(* Logix 5000 project; controller code_tcc vendor 1 type 14 code 106 rev 33.11; software revision 33.01 *)

TASK MainTask (periodic, rate 10 ms, priority 1, watchdog 500 ms) : MainProgram

MODULES
   Local : vendor 1 type 14 code 106 (Compact 0, rev 33.11)
END_MODULES

TYPE raC_UDT_ModbusClientConnection :
STRUCT
   LocalSlot : SINT;   // Local Slot for Ethernet module. For ControlLogix - L8x, EN2T(R) - use the actual module slot. For CompactLogix use slot 0.
   LocalAddress : STR0016;   // Used only for controllers with more than 1 local IP address (5380, 5480). For all others must be blank.
   DestAddress : STR0016;   // The IP address for the Modbus TCP Slave device to connect to
   DestinationPort : DINT;   // Default Modbus is 502
   MSG_Src : SINT[500];   // Placeholder for message source
   MSG_Dest : SINT[500];   // Placeholder for message destination
END_STRUCT
END_TYPE

TYPE raC_UDT_ModbusClientData :
STRUCT
   Coils_0xxx : BOOL[1024];
   DiscInputs_1xxx : BOOL[1024];
   InpRegisters_3xxx : INT[1024];
   HoldRegisters_4xxx : INT[1024];
END_STRUCT
END_TYPE

TYPE raC_UDT_ModbusClientHMI :
STRUCT
   Parameters : raC_UDT_ModbusClientConnection;
   Transaction : raC_UDT_ModbusClientTransaction;
   Index0x : DINT;
   Index1x : DINT;
   Index3x : DINT;
   Index4x : DINT;
   DataValue : INT[65];
   DataAddr : DINT[65];
   TransactionIndex : DINT;
   RemoteAddrStart : DINT;
   RemoteAddrEnd : DINT;
   LocalAddrEnd : DINT;
END_STRUCT
END_TYPE

TYPE raC_UDT_ModbusClientTransaction :
STRUCT
   Enabled : BOOL;   // Enables (1) or disables (0) the transaction
   PollInterval : DINT;   // Time between triggers in milliseconds. Minimum is 80 msec. Anyting below 80 will be set to 1 seconds
   TransType : INT;   // Transaction code for the Modbus Protocol. Acceptable values are 1-Coil Read, 2- Discrete Input read, 3-Holding Register Read, 4-Input Register Read, 5-Write Single Coil, 6-Single Holding Register Write, 15-Multiple Coil Write, 16 Multiple Holding Register Write
   StationID : SINT;   // Station ID ( Unit Identifier). Commonly used if going through a gateway or bridge in which case it is the device address on the other side of the gateway. Other wise leave as 0
   BeginAddress : DINT;   // Beginning address in remote device to read from or write to.
   Count : INT;   // The number of items in remote device to read from or write to.
   LocalAddress : INT;   // Beginning address in in this programs' "_Data" arrays
   TransComplete : BOOL;   // Transaction Complete Flag. Check the TransStat to see if the transaction was successful or if a Modbus exception code was returned.
   TransStat : INT;   // Status result of the transaction. 0 = success, 1 = in process 2 = retry -1 = exception
   Diagnostic : raC_UDT_ModbusClientTransactionDiag;
END_STRUCT
END_TYPE

TYPE raC_UDT_ModbusClientTransactionDiag :
STRUCT
   Request : STR0500;   // Actual buffer used to build the modbus request that is transmited to the remote node.
   ReqBuilt : BOOL;   // Transaction request string is built, clear this if anything is changed in a read operation to rebuild the Request string.
   Overlap : BOOL;   // Transaction is not completing before next trigger
   Overload : BOOL;   // Transaction is not completing because of excessive Overlaps in one or more transactions
   TransID : INT;   // Serial Number of the actual Ethernet Transaction used to match to the appropriate Reply
   TransLastError : INT;   // Last Error on transaction. 0-Success, -2 Network write error, -3 Local write error, -4 Network Read Error, -5 Local Read Error, -6 Connection failed.. -12 Invalid Trans code, -13 Out of data array range.
   IntervalTimer : TIMER;   // IntervalTimer, used to trigger transaction
   NoReplyCounter : COUNTER;   // No Reply Counter
   PendingTimer : TIMER;   // Timing pending requests
END_STRUCT
END_TYPE

TYPE raC_UDT_ModbusConnectParam :   // Parameterss for the OpenConnection Service
STRUCT
   Timeout : DINT;
   DestAddr : STR0032;
END_STRUCT
END_TYPE

TYPE raC_UDT_ModbusCreateParam :
STRUCT
   Type : DINT;   // Type 1-TCP, 2-UDP
   Family : INT;   // Address Family Must be 2
   Port : INT;   // Local Port Number
   Addr : DINT;   // Local IP Address
END_STRUCT
END_TYPE

TYPE STR0008 :
STRUCT
   LEN : DINT;
   DATA : SINT[8];
END_STRUCT
END_TYPE

TYPE STR0016 :
STRUCT
   LEN : DINT;
   DATA : SINT[16];
END_STRUCT
END_TYPE

TYPE STR0032 :
STRUCT
   LEN : DINT;
   DATA : SINT[32];
END_STRUCT
END_TYPE

TYPE STR0500 :
STRUCT
   LEN : DINT;
   DATA : SINT[500];
END_STRUCT
END_TYPE

TYPE STR4096 :
STRUCT
   LEN : DINT;
   DATA : SINT[4096];
END_STRUCT
END_TYPE

ADD_ON_INSTRUCTION raC_Opr_NetModbusTCPClient   (* revision 2.4 0, ExecutePrescan *)
// Modbus TCP Client
// Revision note:
// 2.0.0 Initial Release in AOI format
// 2.0.1 Corrected local IP address logic
// 2.1.0 Corrected Overload and Overlap indicators
// 2.2.0 Changed BeginAddress from INT to DINT, force LocalSlot 0 for CompactLogix
// 2.3.0 HMI interface
// 2.4.0 Improved malformed packet handling
VAR_INPUT
   Inp_Enable : BOOL; {required}
END_VAR
VAR_IN_OUT
   Ref_Connection : raC_UDT_ModbusClientConnection; {required}
   Ref_Transactions : raC_UDT_ModbusClientTransaction[5]; {required}
   Ref_ModbusData : raC_UDT_ModbusClientData; {required}
   Ref_MsgCreate : MESSAGE; {required}
   Ref_MsgConnect : MESSAGE; {required}
   Ref_MsgRead : MESSAGE; {required}
   Ref_MsgWrite : MESSAGE; {required}
   Ref_MsgDelete : MESSAGE; {required}
   Ref_MsgSetAttrSingle : MESSAGE; {required}
END_VAR
VAR_OUTPUT
   Sts_EN : BOOL; {access Read Only, visible}
   Sts_Connected : BOOL; {access Read Only, visible}
   Sts_Faulted : BOOL; {access Read Only, visible}
   Sts_Overlap : BOOL; {access Read Only, visible}
   Sts_Overload : BOOL; {access Read Only, visible}
   Sts_LastError : DINT; {access Read Only}   // The last recorded socket error for this connection. 0 good, -2 Write Error, -4 Read Error, -6 connection failed, -7 Delete all failed, -8 Create Soc failed, -9 Connection failed, -10 connection dropped, -11 error in setting socket parameter. -12 - Enable removed
END_VAR
VAR
   Wrk_MSGStep : DINT; {access None}
   Wrk_CreateReq : raC_UDT_ModbusCreateParam; {access None}
   Wrk_Instance : DINT; {access None}
   Wrk_ConnectReq : raC_UDT_ModbusConnectParam; {access None}
   Wrk_PortStr : STR0016 := '?port='; {access None}
   Wrk_TempStr : STR0016; {access None}
   Wrk_RetryTimer : TIMER := (PRE := 5000); {access None}
   Wrk_MSGRead_SRC : DINT[2]; {access None}   // User for MSG Read Source
   Wrk_TempString : STR0500; {access None}
   Wrk_Main_Read_Buffer : STR4096; {access None}
   Wrk_WrIndex : DINT; {access None}
   Wrk_TransactionTriggers : BOOL[32]; {access None}
   Wrk_BRS : raC_Tec_NetModbusTCPClient_BuildReqStr; {access None}
   Wrk_IDCounter : DINT; {access None}
   Wrk_WriteNow : BOOL[32]; {access None}   // Transmit Request Flags
   Wrk_TempDINT : DINT; {access None}
   Wrk_AdditionalLen : INT; {access None}
   Wrk_ModbusTransID : INT; {access None}
   Wrk_AdditionaLenRead : INT; {access None}
   Wrk_ModbusCmdLen : INT; {access None}
   Wrk_ModbusPacket : STR0500; {access None}
   Wrk_DataReceived : BOOL; {access None}
   Wrk_CmdFromReadPacket : DINT; {access None}
   Wrk_ModbusID : STR0008; {access None}
   Wrk_AdditionalLen1 : INT; {access None}
   Wrk_ModbusCmdTemp : INT; {access None}
   Wrk_ModbusUnit : STR0008; {access None}
   Wrk_ModbusBytes : DINT; {access None}
   Wrk_ModbusCmdString : STR0500; {access None}
   Wrk_CWR : raC_Tec_NetModbusTCPClient_ChkWrReply; {access None}
   Wrk_RSB : raC_Tec_NetModbusTCPClient_RespStrBit; {access None}
   Wrk_TransIndex : DINT; {access None}
   Wrk_TimerIndex : DINT; {access None}
   Wrk_ArraySize : DINT; {access None}
   Wrk_LastTransaction : DINT; {access None}
   Wrk_RSW : raC_Tec_NetModbusTCPClient_RespStrWord; {access None}
   Wrk_TempOctet : DINT[4]; {access None}
   Wrk_TempStrOctet : STR0008; {access None}
   Wrk_TempStrOctetlen : DINT; {access None}
   Wrk_TempIPStr : STR0016; {access None}
   Wrk_TempInt : DINT; {access None}
   Wrk_ClrReqIndex : DINT; {access None}
   Wrk_StepLockTimer : TIMER := (PRE := 10000); {access None}
   Wrk_Controller_Name : SINT[33]; {access None}
   Wrk_Controller_Type : DINT; {access None}
   Wrk_InitCompleted : BOOL; {access None}
   Inf_Lib : STR0016; {access Read Only}
   Inf_Type : STR0032; {access Read Only}
   Inf_Version : STR0016; {access Read Only}
   HMI_Tab : DINT;
   Wrk_tempHMItransaction : DINT; {access None}
   Wrk_HMITransactionValid : BOOL; {access None}
   wrk_FAL_Addr : CONTROL := (LEN := 64); {access None}
   wrk_LoopIndex : DINT; {access None}
   wrk_AddrIndex : DINT; {access None}
   HMI : raC_UDT_ModbusClientHMI;
   Wrk_OLindex : DINT; {access None}
   Wrk_OverloadStatus : BOOL; {access None}
   Wrk_OverlapStatus : BOOL; {access None}
END_VAR

ROUTINE Logic   (* ladder *)
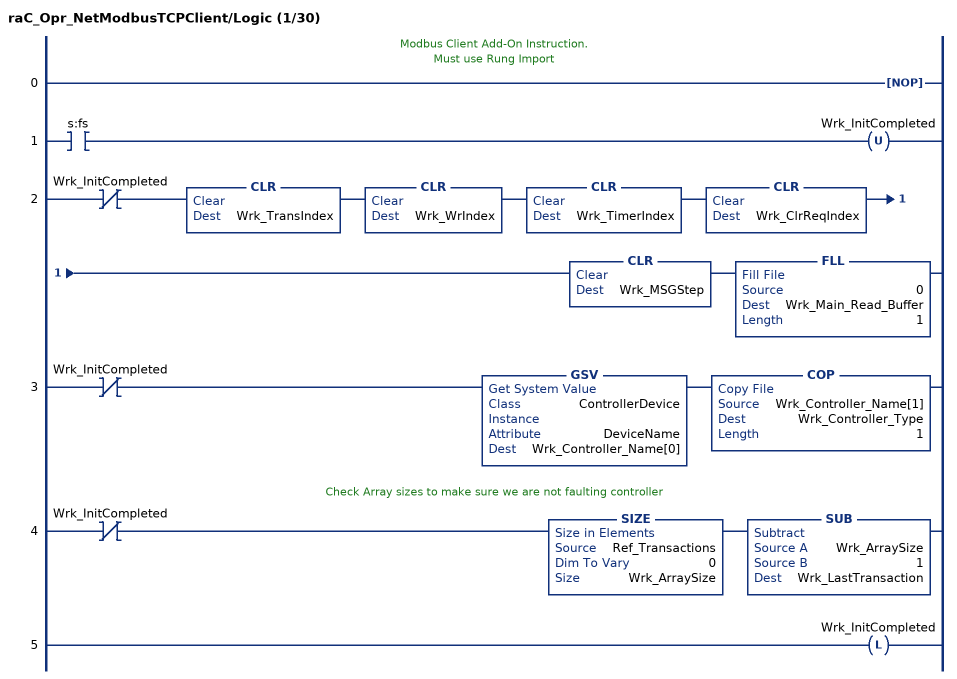
   // Modbus Client Add-On Instruction.
   // Must use Rung Import
   0: NOP();
   1: XIC(s:fs)OTU(Wrk_InitCompleted);
   2: XIO(Wrk_InitCompleted)CLR(Wrk_TransIndex)CLR(Wrk_WrIndex)CLR(Wrk_TimerIndex)CLR(Wrk_ClrReqIndex)CLR(Wrk_MSGStep)FLL(0,Wrk_Main_Read_Buffer,1);
   3: XIO(Wrk_InitCompleted)GSV(ControllerDevice,,DeviceName,Wrk_Controller_Name[0])COP(Wrk_Controller_Name[1],Wrk_Controller_Type,1);
   // Check Array sizes to make sure we are not faulting controller
   4: XIO(Wrk_InitCompleted)SIZE(Ref_Transactions,0,Wrk_ArraySize)SUB(Wrk_ArraySize,1,Wrk_LastTransaction);
   5: OTL(Wrk_InitCompleted);
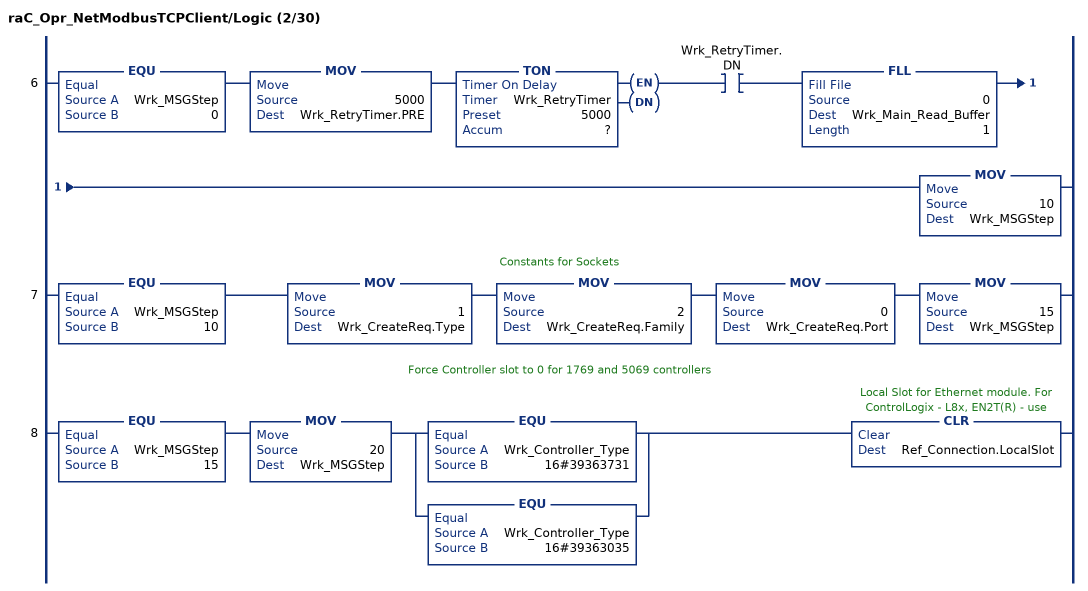
   6: EQU(Wrk_MSGStep,0)MOV(5000,Wrk_RetryTimer.PRE)TON(Wrk_RetryTimer,?,?)XIC(Wrk_RetryTimer.DN)FLL(0,Wrk_Main_Read_Buffer,1)MOV(10,Wrk_MSGStep);
   // Constants for Sockets
   7: EQU(Wrk_MSGStep,10)MOV(1,Wrk_CreateReq.Type)MOV(2,Wrk_CreateReq.Family)MOV(0,Wrk_CreateReq.Port)MOV(15,Wrk_MSGStep);
   // Force Controller slot to 0 for 1769 and 5069 controllers
   8: EQU(Wrk_MSGStep,15)MOV(20,Wrk_MSGStep)[EQU(Wrk_Controller_Type,16#39363731) ,EQU(Wrk_Controller_Type,16#39363035) ]CLR(Ref_Connection.LocalSlot);
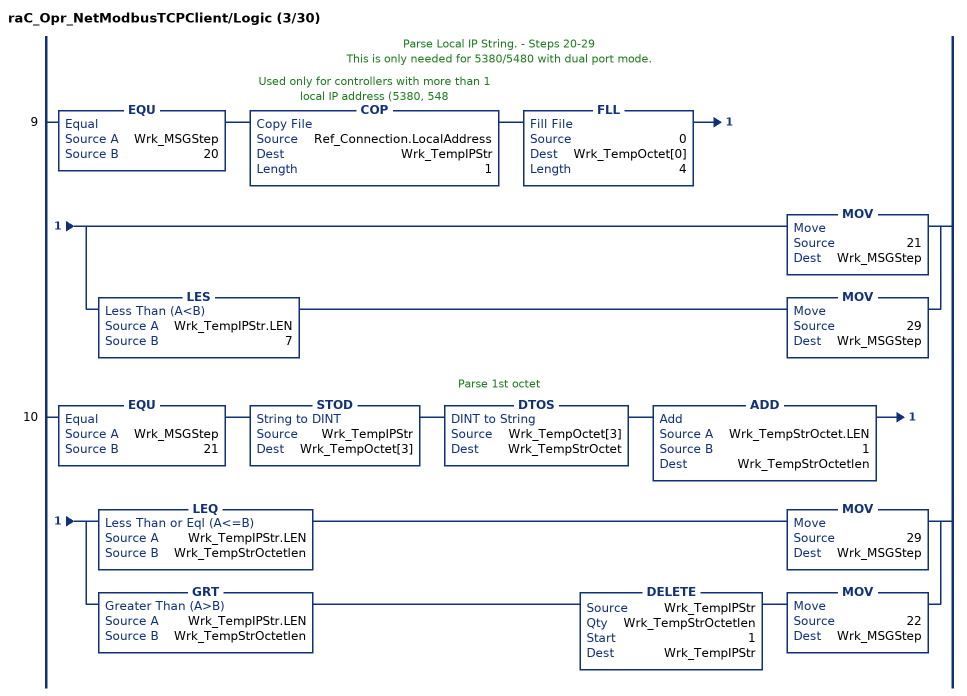
   // Parse Local IP String. - Steps 20-29
   // This is only needed for 5380/5480 with dual port mode.
   9: EQU(Wrk_MSGStep,20)COP(Ref_Connection.LocalAddress,Wrk_TempIPStr,1)FLL(0,Wrk_TempOctet[0],4)[MOV(21,Wrk_MSGStep) ,LES(Wrk_TempIPStr.LEN,7) MOV(29,Wrk_MSGStep) ];
   // Parse 1st octet
   10: EQU(Wrk_MSGStep,21)STOD(Wrk_TempIPStr,Wrk_TempOctet[3])DTOS(Wrk_TempOctet[3],Wrk_TempStrOctet)ADD(Wrk_TempStrOctet.LEN,1,Wrk_TempStrOctetlen)[LEQ(Wrk_TempIPStr.LEN,Wrk_TempStrOctetlen) MOV(29,Wrk_MSGStep) ,GRT(Wrk_TempIPStr.LEN,Wrk_TempStrOctetlen) DELETE(Wrk_TempIPStr,Wrk_TempStrOctetlen,1,Wrk_TempIPStr) MOV(22,Wrk_MSGStep) ];
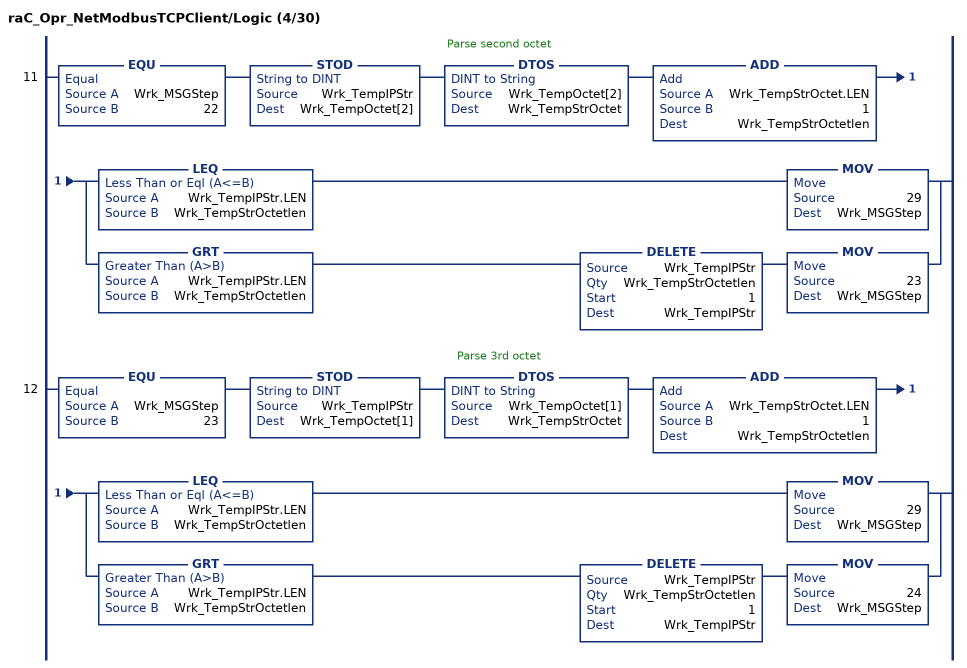
   // Parse second octet
   11: EQU(Wrk_MSGStep,22)STOD(Wrk_TempIPStr,Wrk_TempOctet[2])DTOS(Wrk_TempOctet[2],Wrk_TempStrOctet)ADD(Wrk_TempStrOctet.LEN,1,Wrk_TempStrOctetlen)[LEQ(Wrk_TempIPStr.LEN,Wrk_TempStrOctetlen) MOV(29,Wrk_MSGStep) ,GRT(Wrk_TempIPStr.LEN,Wrk_TempStrOctetlen) DELETE(Wrk_TempIPStr,Wrk_TempStrOctetlen,1,Wrk_TempIPStr) MOV(23,Wrk_MSGStep) ];
   // Parse 3rd octet
   12: EQU(Wrk_MSGStep,23)STOD(Wrk_TempIPStr,Wrk_TempOctet[1])DTOS(Wrk_TempOctet[1],Wrk_TempStrOctet)ADD(Wrk_TempStrOctet.LEN,1,Wrk_TempStrOctetlen)[LEQ(Wrk_TempIPStr.LEN,Wrk_TempStrOctetlen) MOV(29,Wrk_MSGStep) ,GRT(Wrk_TempIPStr.LEN,Wrk_TempStrOctetlen) DELETE(Wrk_TempIPStr,Wrk_TempStrOctetlen,1,Wrk_TempIPStr) MOV(24,Wrk_MSGStep) ];
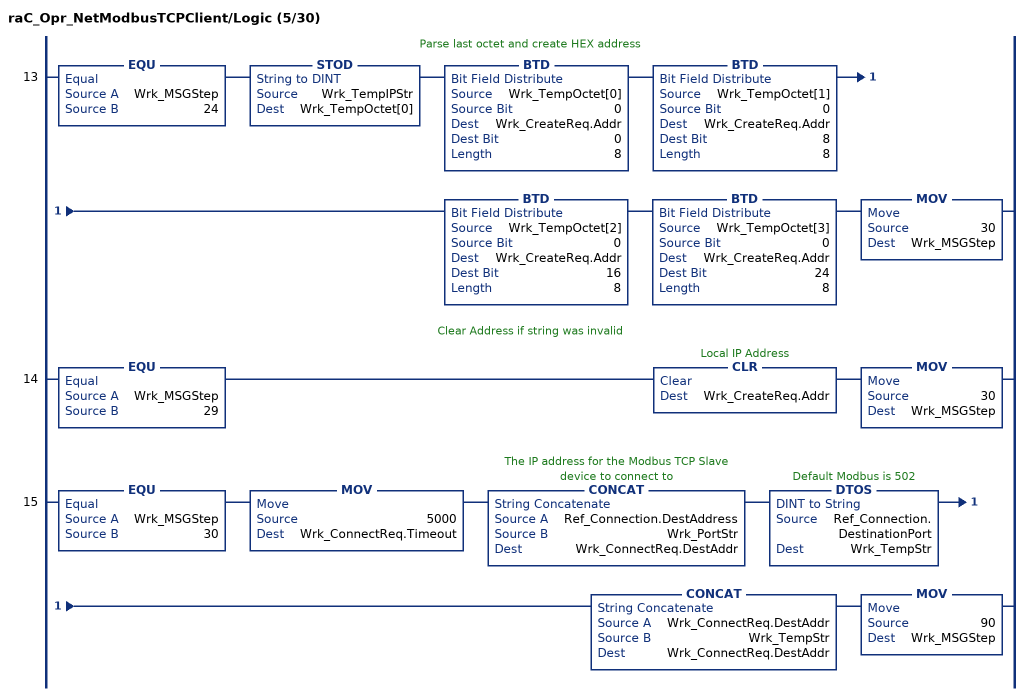
   // Parse last octet and create HEX address
   13: EQU(Wrk_MSGStep,24)STOD(Wrk_TempIPStr,Wrk_TempOctet[0])BTD(Wrk_TempOctet[0],0,Wrk_CreateReq.Addr,0,8)BTD(Wrk_TempOctet[1],0,Wrk_CreateReq.Addr,8,8)BTD(Wrk_TempOctet[2],0,Wrk_CreateReq.Addr,16,8)BTD(Wrk_TempOctet[3],0,Wrk_CreateReq.Addr,24,8)MOV(30,Wrk_MSGStep);
   // Clear Address if string was invalid
   14: EQU(Wrk_MSGStep,29)CLR(Wrk_CreateReq.Addr)MOV(30,Wrk_MSGStep);
   15: EQU(Wrk_MSGStep,30)MOV(5000,Wrk_ConnectReq.Timeout)CONCAT(Ref_Connection.DestAddress,Wrk_PortStr,Wrk_ConnectReq.DestAddr)DTOS(Ref_Connection.DestinationPort,Wrk_TempStr)CONCAT(Wrk_ConnectReq.DestAddr,Wrk_TempStr,Wrk_ConnectReq.DestAddr)MOV(90,Wrk_MSGStep);
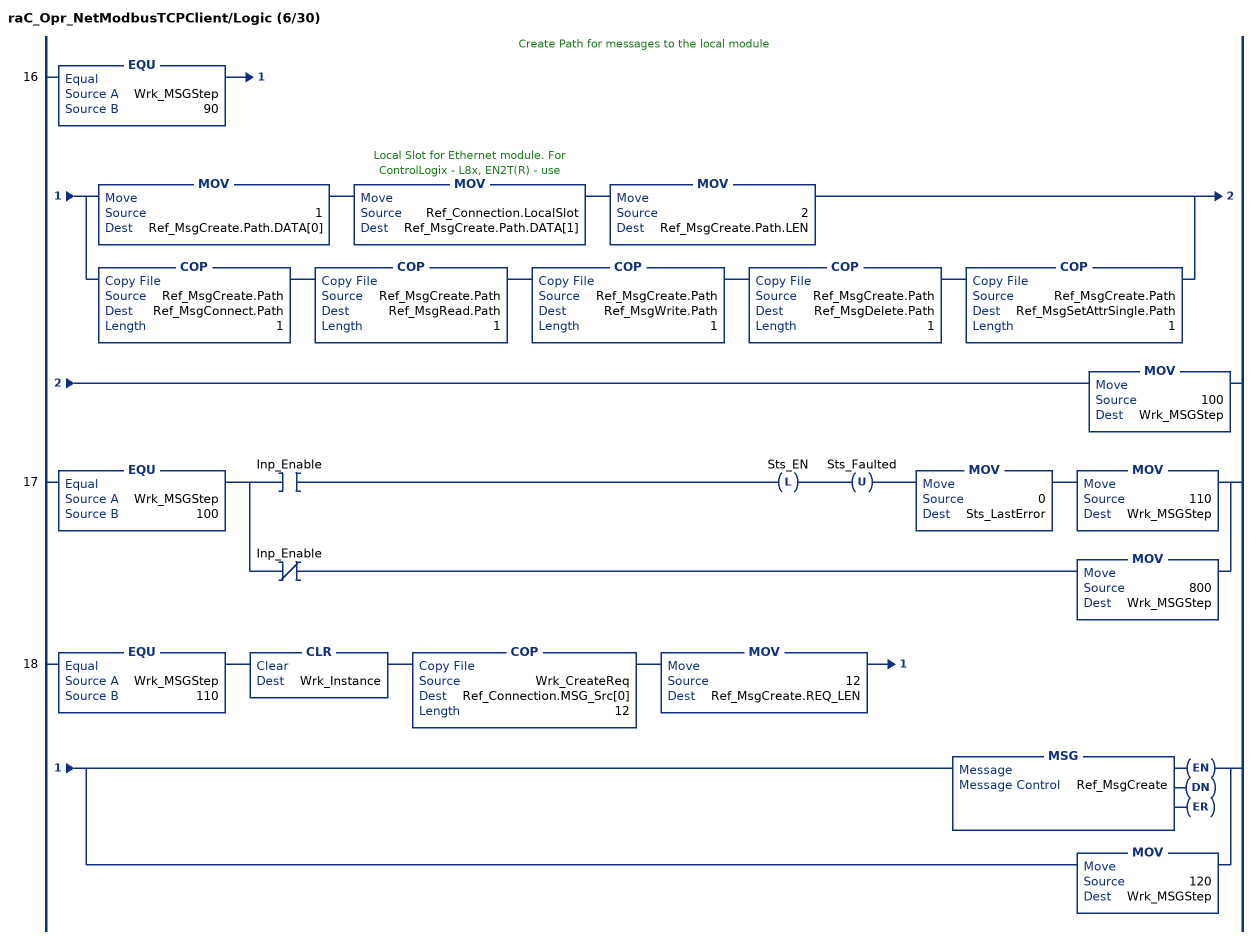
   // Create Path for messages to the local module
   16: EQU(Wrk_MSGStep,90)[MOV(1,Ref_MsgCreate.Path.DATA[0]) MOV(Ref_Connection.LocalSlot,Ref_MsgCreate.Path.DATA[1]) MOV(2,Ref_MsgCreate.Path.LEN) ,COP(Ref_MsgCreate.Path,Ref_MsgConnect.Path,1) COP(Ref_MsgCreate.Path,Ref_MsgRead.Path,1) COP(Ref_MsgCreate.Path,Ref_MsgWrite.Path,1) COP(Ref_MsgCreate.Path,Ref_MsgDelete.Path,1) COP(Ref_MsgCreate.Path,Ref_MsgSetAttrSingle.Path,1) ]MOV(100,Wrk_MSGStep);
   17: EQU(Wrk_MSGStep,100)[XIC(Inp_Enable) OTL(Sts_EN) OTU(Sts_Faulted) MOV(0,Sts_LastError) MOV(110,Wrk_MSGStep) ,XIO(Inp_Enable) MOV(800,Wrk_MSGStep) ];
   18: EQU(Wrk_MSGStep,110)CLR(Wrk_Instance)COP(Wrk_CreateReq,Ref_Connection.MSG_Src[0],12)MOV(12,Ref_MsgCreate.REQ_LEN)[MSG(Ref_MsgCreate) ,MOV(120,Wrk_MSGStep) ];
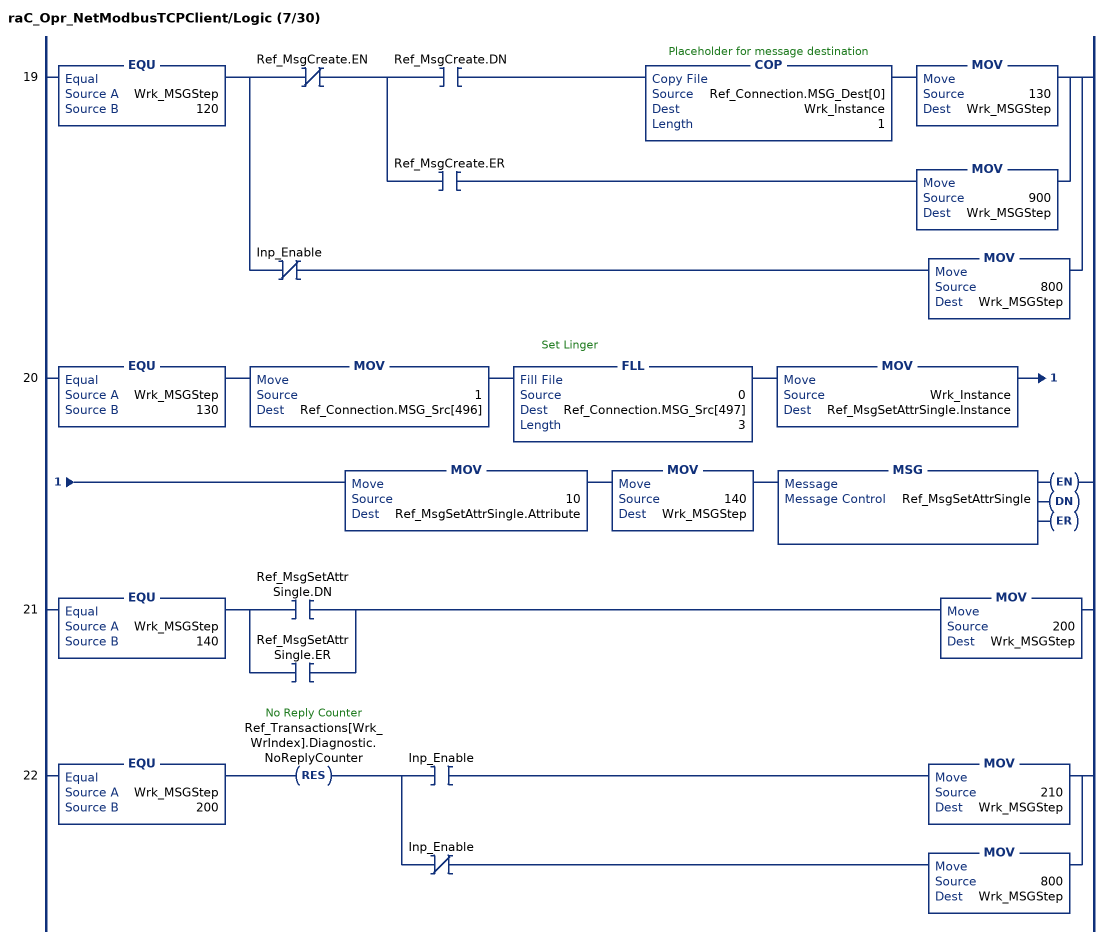
   19: EQU(Wrk_MSGStep,120)[XIO(Ref_MsgCreate.EN) [XIC(Ref_MsgCreate.DN) COP(Ref_Connection.MSG_Dest[0],Wrk_Instance,1) MOV(130,Wrk_MSGStep) ,XIC(Ref_MsgCreate.ER) MOV(900,Wrk_MSGStep) ] ,XIO(Inp_Enable) MOV(800,Wrk_MSGStep) ];
   // Set Linger
   20: EQU(Wrk_MSGStep,130)MOV(1,Ref_Connection.MSG_Src[496])FLL(0,Ref_Connection.MSG_Src[497],3)MOV(Wrk_Instance,Ref_MsgSetAttrSingle.Instance)MOV(10,Ref_MsgSetAttrSingle.Attribute)MOV(140,Wrk_MSGStep)MSG(Ref_MsgSetAttrSingle);
   21: EQU(Wrk_MSGStep,140)[XIC(Ref_MsgSetAttrSingle.DN) ,XIC(Ref_MsgSetAttrSingle.ER) ]MOV(200,Wrk_MSGStep);
   22: EQU(Wrk_MSGStep,200)RES(Ref_Transactions[Wrk_WrIndex].Diagnostic.NoReplyCounter)[XIC(Inp_Enable) MOV(210,Wrk_MSGStep) ,XIO(Inp_Enable) MOV(800,Wrk_MSGStep) ];
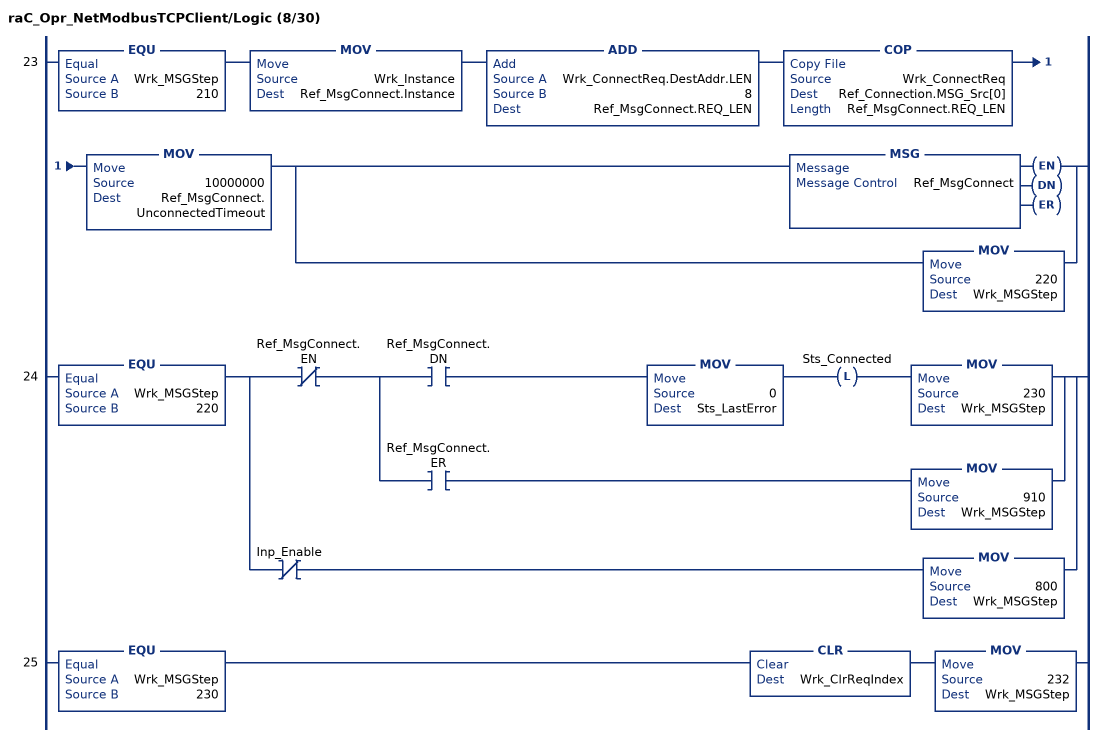
   23: EQU(Wrk_MSGStep,210)MOV(Wrk_Instance,Ref_MsgConnect.Instance)ADD(Wrk_ConnectReq.DestAddr.LEN,8,Ref_MsgConnect.REQ_LEN)COP(Wrk_ConnectReq,Ref_Connection.MSG_Src[0],Ref_MsgConnect.REQ_LEN)MOV(10000000,Ref_MsgConnect.UnconnectedTimeout)[MSG(Ref_MsgConnect) ,MOV(220,Wrk_MSGStep) ];
   24: EQU(Wrk_MSGStep,220)[XIO(Ref_MsgConnect.EN) [XIC(Ref_MsgConnect.DN) MOV(0,Sts_LastError) OTL(Sts_Connected) MOV(230,Wrk_MSGStep) ,XIC(Ref_MsgConnect.ER) MOV(910,Wrk_MSGStep) ] ,XIO(Inp_Enable) MOV(800,Wrk_MSGStep) ];
   25: EQU(Wrk_MSGStep,230)CLR(Wrk_ClrReqIndex)MOV(232,Wrk_MSGStep);
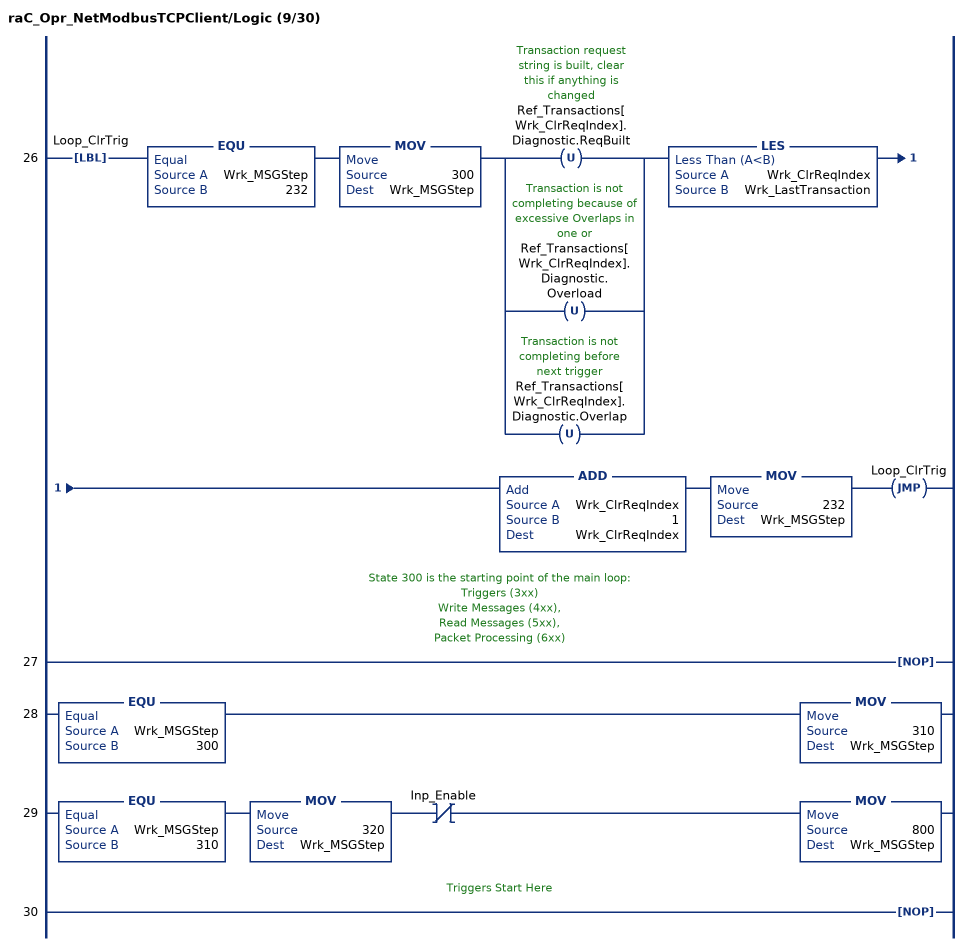
   26: LBL(Loop_ClrTrig)EQU(Wrk_MSGStep,232)MOV(300,Wrk_MSGStep)[OTU(Ref_Transactions[Wrk_ClrReqIndex].Diagnostic.ReqBuilt) ,OTU(Ref_Transactions[Wrk_ClrReqIndex].Diagnostic.Overload) ,OTU(Ref_Transactions[Wrk_ClrReqIndex].Diagnostic.Overlap) ]LES(Wrk_ClrReqIndex,Wrk_LastTransaction)ADD(Wrk_ClrReqIndex,1,Wrk_ClrReqIndex)MOV(232,Wrk_MSGStep)JMP(Loop_ClrTrig);
   // State 300 is the starting point of the main loop:
   // Triggers (3xx)
   // Write Messages (4xx),
   // Read Messages (5xx),
   // Packet Processing (6xx)
   27: NOP();
   28: EQU(Wrk_MSGStep,300)MOV(310,Wrk_MSGStep);
   29: EQU(Wrk_MSGStep,310)MOV(320,Wrk_MSGStep)XIO(Inp_Enable)MOV(800,Wrk_MSGStep);
   // Triggers Start Here
   30: NOP();
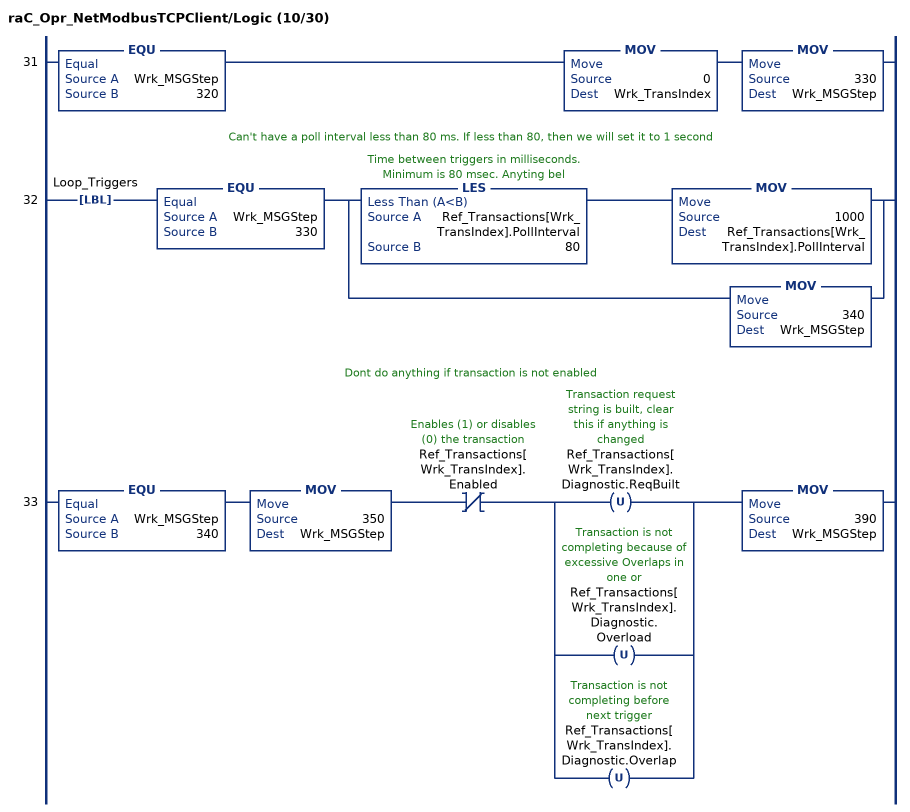
   31: EQU(Wrk_MSGStep,320)MOV(0,Wrk_TransIndex)MOV(330,Wrk_MSGStep);
   // Can't have a poll interval less than 80 ms. If less than 80, then we will set it to 1 second
   32: LBL(Loop_Triggers)EQU(Wrk_MSGStep,330)[LES(Ref_Transactions[Wrk_TransIndex].PollInterval,80) MOV(1000,Ref_Transactions[Wrk_TransIndex].PollInterval) ,MOV(340,Wrk_MSGStep) ];
   // Dont do anything if transaction is not enabled
   33: EQU(Wrk_MSGStep,340)MOV(350,Wrk_MSGStep)XIO(Ref_Transactions[Wrk_TransIndex].Enabled)[OTU(Ref_Transactions[Wrk_TransIndex].Diagnostic.ReqBuilt) ,OTU(Ref_Transactions[Wrk_TransIndex].Diagnostic.Overload) ,OTU(Ref_Transactions[Wrk_TransIndex].Diagnostic.Overlap) ]MOV(390,Wrk_MSGStep);
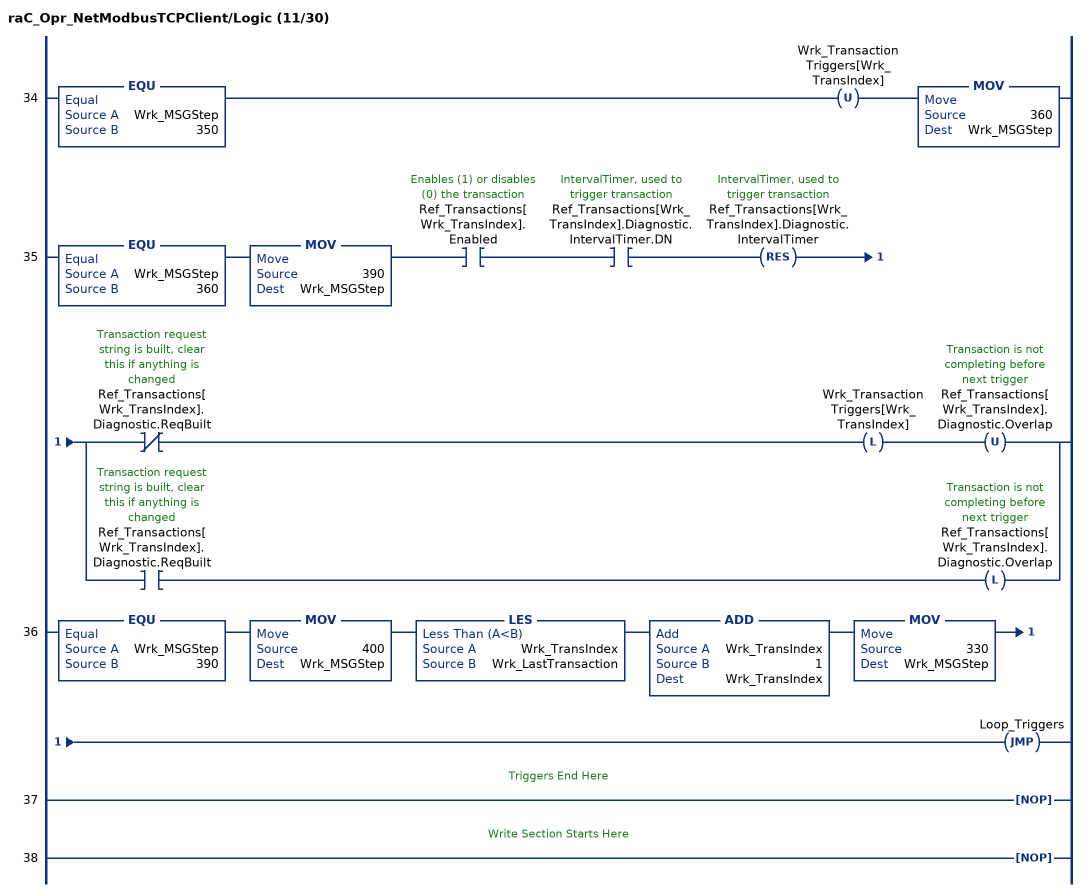
   34: EQU(Wrk_MSGStep,350)OTU(Wrk_TransactionTriggers[Wrk_TransIndex])MOV(360,Wrk_MSGStep);
   35: EQU(Wrk_MSGStep,360)MOV(390,Wrk_MSGStep)XIC(Ref_Transactions[Wrk_TransIndex].Enabled)XIC(Ref_Transactions[Wrk_TransIndex].Diagnostic.IntervalTimer.DN)RES(Ref_Transactions[Wrk_TransIndex].Diagnostic.IntervalTimer)[XIO(Ref_Transactions[Wrk_TransIndex].Diagnostic.ReqBuilt) OTL(Wrk_TransactionTriggers[Wrk_TransIndex]) OTU(Ref_Transactions[Wrk_TransIndex].Diagnostic.Overlap) ,XIC(Ref_Transactions[Wrk_TransIndex].Diagnostic.ReqBuilt) OTL(Ref_Transactions[Wrk_TransIndex].Diagnostic.Overlap) ];
   36: EQU(Wrk_MSGStep,390)MOV(400,Wrk_MSGStep)LES(Wrk_TransIndex,Wrk_LastTransaction)ADD(Wrk_TransIndex,1,Wrk_TransIndex)MOV(330,Wrk_MSGStep)JMP(Loop_Triggers);
   // Triggers End Here
   37: NOP();
   // Write Section Starts Here
   38: NOP();
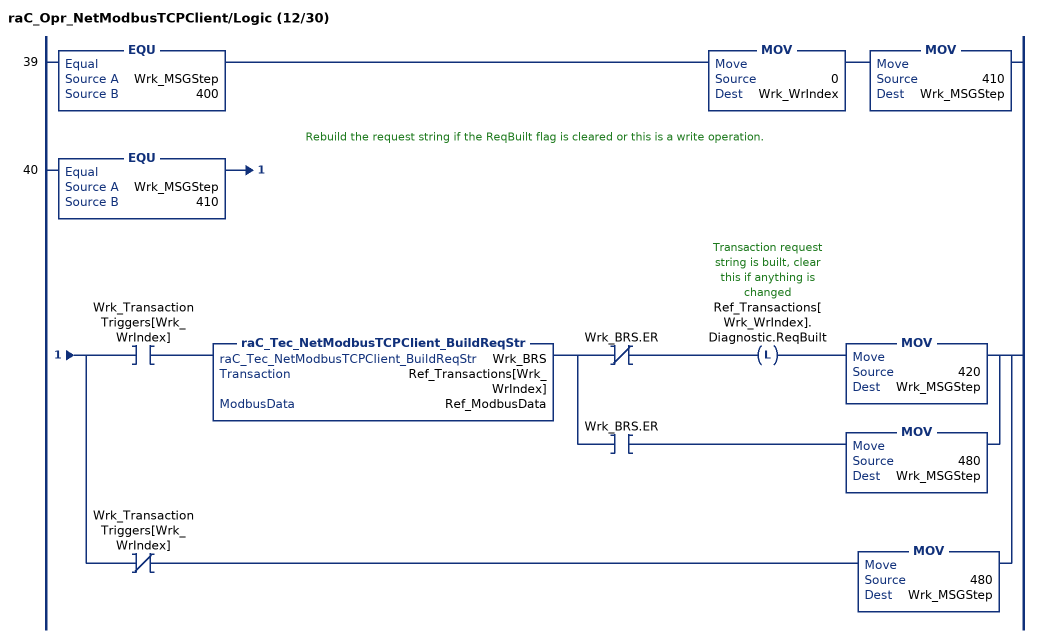
   39: EQU(Wrk_MSGStep,400)MOV(0,Wrk_WrIndex)MOV(410,Wrk_MSGStep);
   // Rebuild the request string if the ReqBuilt flag is cleared or this is a write operation.
   40: EQU(Wrk_MSGStep,410)[XIC(Wrk_TransactionTriggers[Wrk_WrIndex]) raC_Tec_NetModbusTCPClient_BuildReqStr(Wrk_BRS,Ref_Transactions[Wrk_WrIndex],Ref_ModbusData) [XIO(Wrk_BRS.ER) OTL(Ref_Transactions[Wrk_WrIndex].Diagnostic.ReqBuilt) MOV(420,Wrk_MSGStep) ,XIC(Wrk_BRS.ER) MOV(480,Wrk_MSGStep) ] ,XIO(Wrk_TransactionTriggers[Wrk_WrIndex]) MOV(480,Wrk_MSGStep) ];
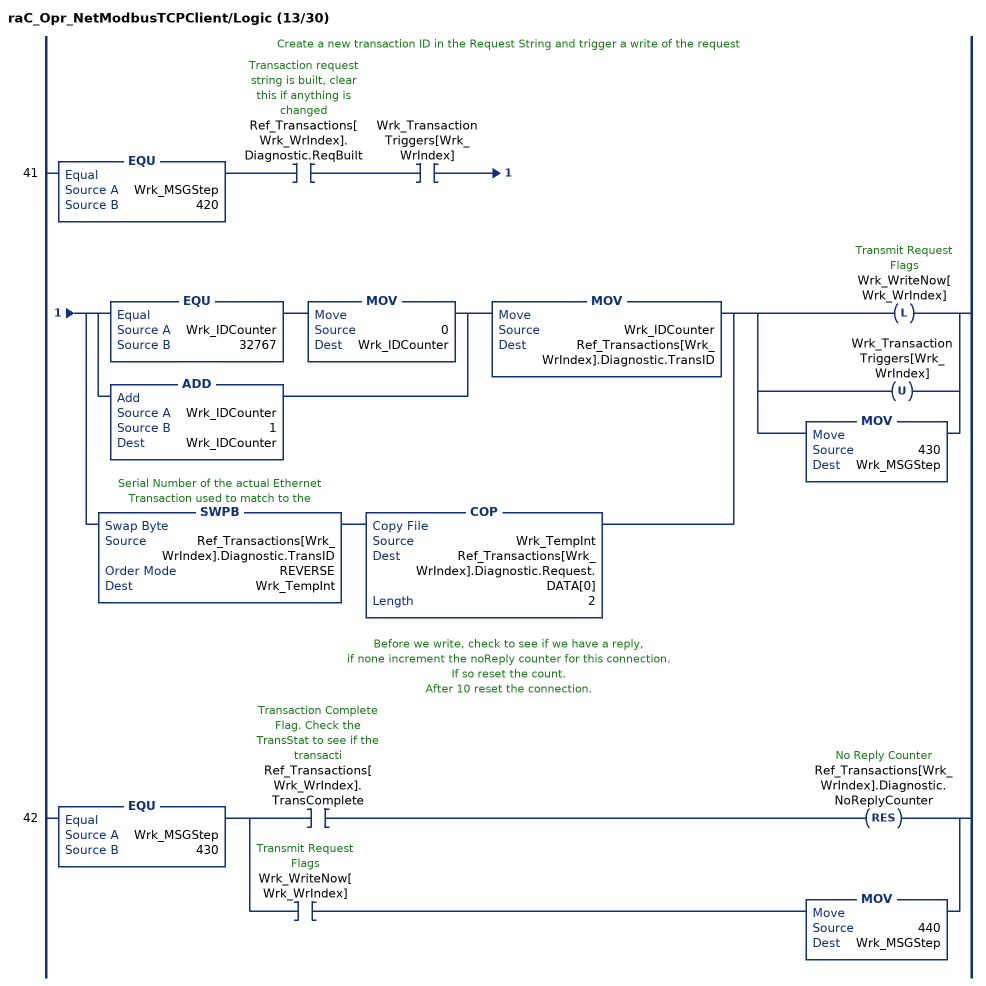
   // Create a new transaction ID in the Request String and trigger a write of the request
   41: EQU(Wrk_MSGStep,420)XIC(Ref_Transactions[Wrk_WrIndex].Diagnostic.ReqBuilt)XIC(Wrk_TransactionTriggers[Wrk_WrIndex])[[EQU(Wrk_IDCounter,32767) MOV(0,Wrk_IDCounter) ,ADD(Wrk_IDCounter,1,Wrk_IDCounter) ] MOV(Wrk_IDCounter,Ref_Transactions[Wrk_WrIndex].Diagnostic.TransID) ,SWPB(Ref_Transactions[Wrk_WrIndex].Diagnostic.TransID,REVERSE,Wrk_TempInt) COP(Wrk_TempInt,Ref_Transactions[Wrk_WrIndex].Diagnostic.Request.DATA[0],2) ][OTL(Wrk_WriteNow[Wrk_WrIndex]) ,OTU(Wrk_TransactionTriggers[Wrk_WrIndex]) ,MOV(430,Wrk_MSGStep) ];
   // Before we write, check to see if we have a reply,
   // if none increment the noReply counter for this connection.
   // If so reset the count.
   // After 10 reset the connection.
   42: EQU(Wrk_MSGStep,430)[XIC(Ref_Transactions[Wrk_WrIndex].TransComplete) RES(Ref_Transactions[Wrk_WrIndex].Diagnostic.NoReplyCounter) ,XIC(Wrk_WriteNow[Wrk_WrIndex]) MOV(440,Wrk_MSGStep) ];
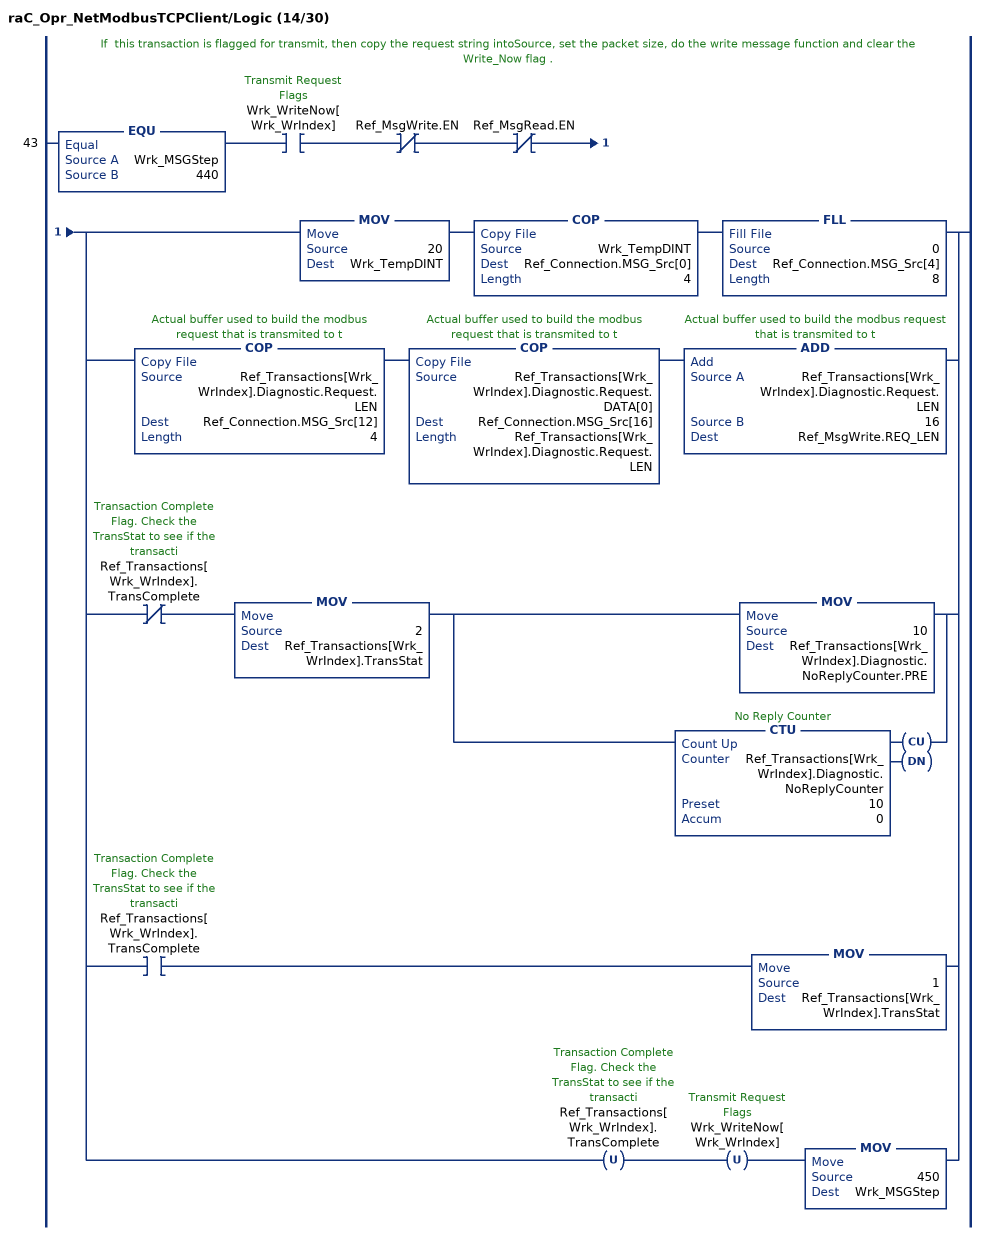
   // If  this transaction is flagged for transmit, then copy the request string intoSource, set the packet size, do the write message function and clear the Write_Now flag .
   43: EQU(Wrk_MSGStep,440)XIC(Wrk_WriteNow[Wrk_WrIndex])XIO(Ref_MsgWrite.EN)XIO(Ref_MsgRead.EN)[MOV(20,Wrk_TempDINT) COP(Wrk_TempDINT,Ref_Connection.MSG_Src[0],4) FLL(0,Ref_Connection.MSG_Src[4],8) ,COP(Ref_Transactions[Wrk_WrIndex].Diagnostic.Request.LEN,Ref_Connection.MSG_Src[12],4) COP(Ref_Transactions[Wrk_WrIndex].Diagnostic.Request.DATA[0],Ref_Connection.MSG_Src[16],Ref_Transactions[Wrk_WrIndex].Diagnostic.Request.LEN) ADD(Ref_Transactions[Wrk_WrIndex].Diagnostic.Request.LEN,16,Ref_MsgWrite.REQ_LEN) ,XIO(Ref_Transactions[Wrk_WrIndex].TransComplete) MOV(2,Ref_Transactions[Wrk_WrIndex].TransStat) [MOV(10,Ref_Transactions[Wrk_WrIndex].Diagnostic.NoReplyCounter.PRE) ,CTU(Ref_Transactions[Wrk_WrIndex].Diagnostic.NoReplyCounter,10,0) ] ,XIC(Ref_Transactions[Wrk_WrIndex].TransComplete) MOV(1,Ref_Transactions[Wrk_WrIndex].TransStat) ,OTU(Ref_Transactions[Wrk_WrIndex].TransComplete) OTU(Wrk_WriteNow[Wrk_WrIndex]) MOV(450,Wrk_MSGStep) ];
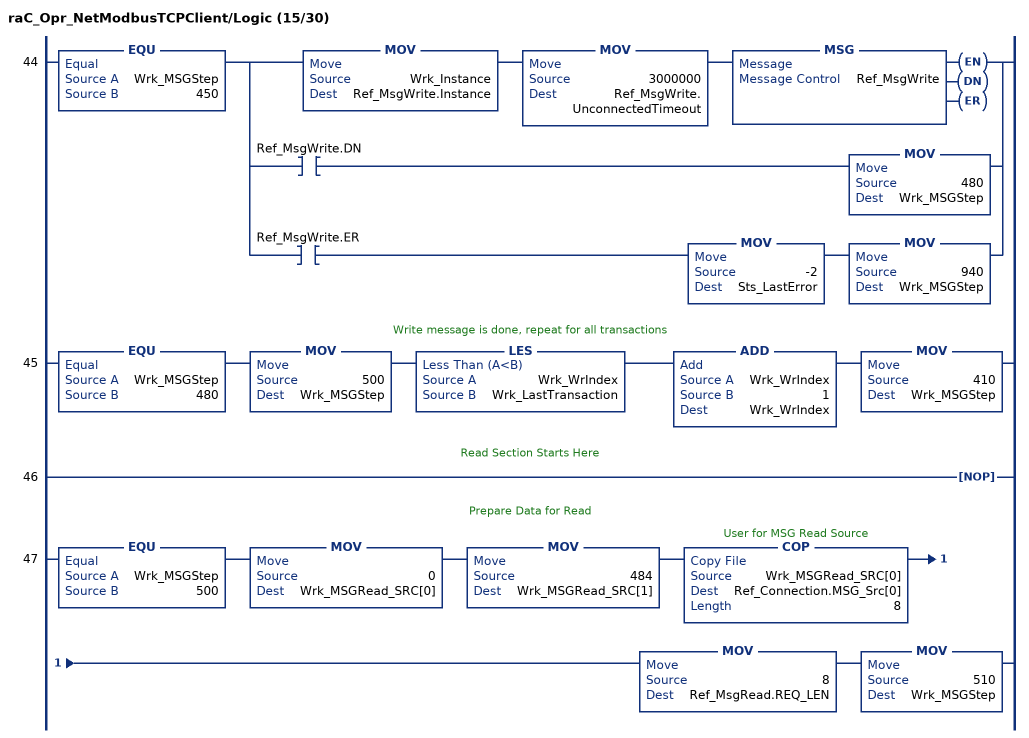
   44: EQU(Wrk_MSGStep,450)[MOV(Wrk_Instance,Ref_MsgWrite.Instance) MOV(3000000,Ref_MsgWrite.UnconnectedTimeout) MSG(Ref_MsgWrite) ,XIC(Ref_MsgWrite.DN) MOV(480,Wrk_MSGStep) ,XIC(Ref_MsgWrite.ER) MOV(-2,Sts_LastError) MOV(940,Wrk_MSGStep) ];
   // Write message is done, repeat for all transactions
   45: EQU(Wrk_MSGStep,480)MOV(500,Wrk_MSGStep)LES(Wrk_WrIndex,Wrk_LastTransaction)ADD(Wrk_WrIndex,1,Wrk_WrIndex)MOV(410,Wrk_MSGStep);
   // Read Section Starts Here
   46: NOP();
   // Prepare Data for Read
   47: EQU(Wrk_MSGStep,500)MOV(0,Wrk_MSGRead_SRC[0])MOV(484,Wrk_MSGRead_SRC[1])COP(Wrk_MSGRead_SRC[0],Ref_Connection.MSG_Src[0],8)MOV(8,Ref_MsgRead.REQ_LEN)MOV(510,Wrk_MSGStep);
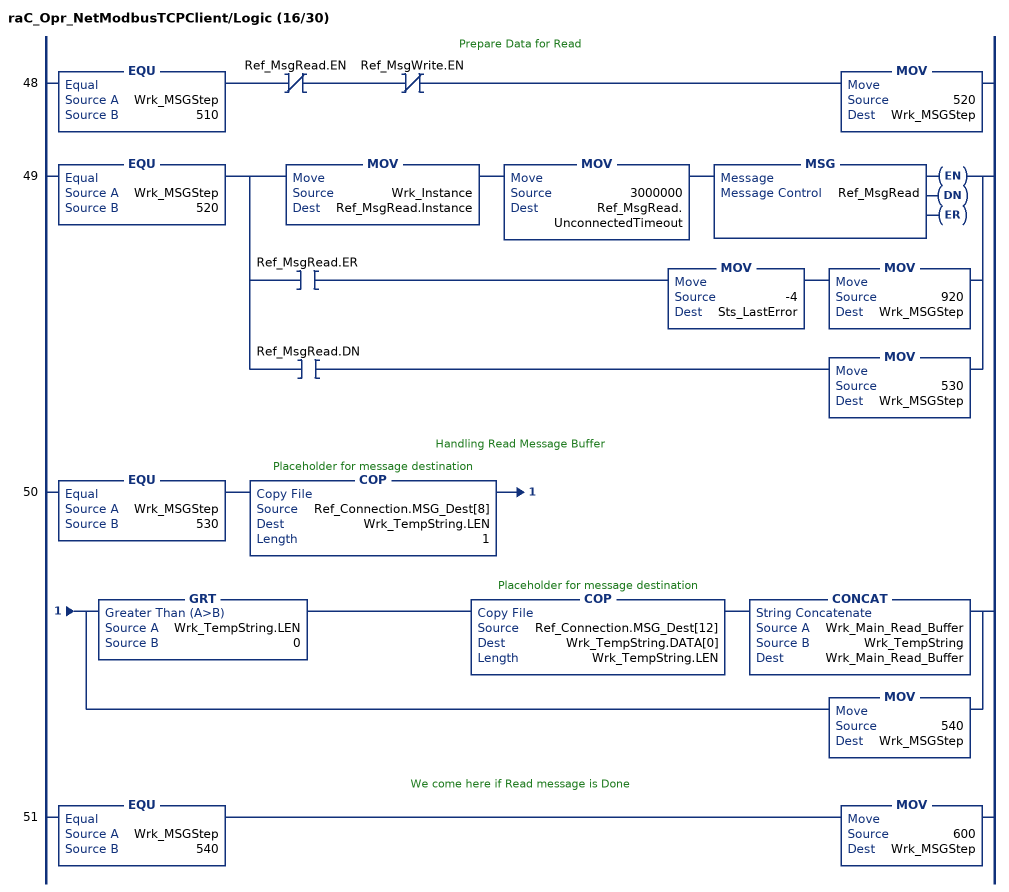
   // Prepare Data for Read
   48: EQU(Wrk_MSGStep,510)XIO(Ref_MsgRead.EN)XIO(Ref_MsgWrite.EN)MOV(520,Wrk_MSGStep);
   49: EQU(Wrk_MSGStep,520)[MOV(Wrk_Instance,Ref_MsgRead.Instance) MOV(3000000,Ref_MsgRead.UnconnectedTimeout) MSG(Ref_MsgRead) ,XIC(Ref_MsgRead.ER) MOV(-4,Sts_LastError) MOV(920,Wrk_MSGStep) ,XIC(Ref_MsgRead.DN) MOV(530,Wrk_MSGStep) ];
   // Handling Read Message Buffer
   50: EQU(Wrk_MSGStep,530)COP(Ref_Connection.MSG_Dest[8],Wrk_TempString.LEN,1)[GRT(Wrk_TempString.LEN,0) COP(Ref_Connection.MSG_Dest[12],Wrk_TempString.DATA[0],Wrk_TempString.LEN) CONCAT(Wrk_Main_Read_Buffer,Wrk_TempString,Wrk_Main_Read_Buffer) ,MOV(540,Wrk_MSGStep) ];
   // We come here if Read message is Done
   51: EQU(Wrk_MSGStep,540)MOV(600,Wrk_MSGStep);
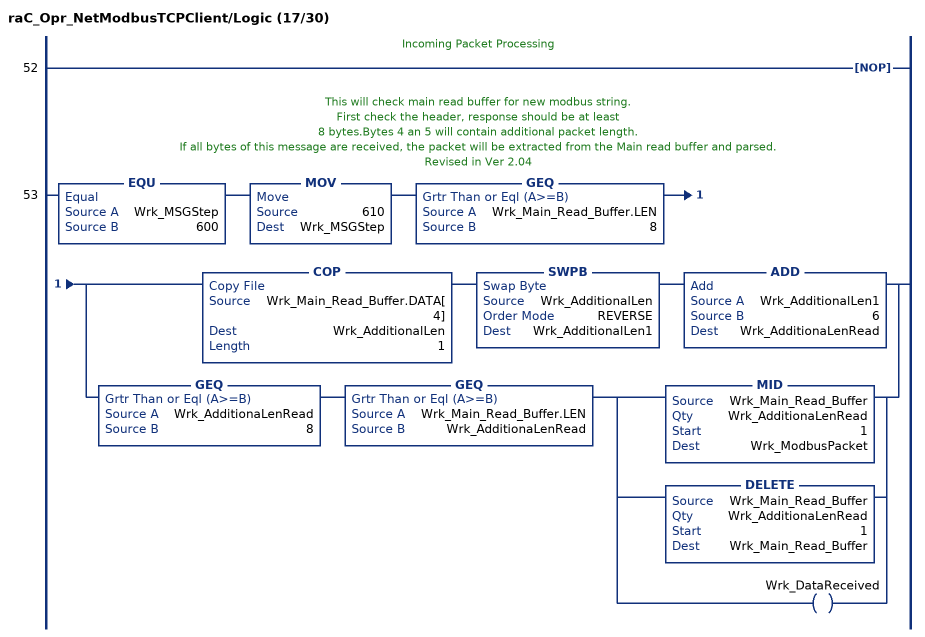
   // Incoming Packet Processing
   52: NOP();
   // This will check main read buffer for new modbus string.
   // First check the header, response should be at least
   // 8 bytes.Bytes 4 an 5 will contain additional packet length.
   // If all bytes of this message are received, the packet will be extracted from the Main read buffer and parsed.
   // Revised in Ver 2.04
   53: EQU(Wrk_MSGStep,600)MOV(610,Wrk_MSGStep)GEQ(Wrk_Main_Read_Buffer.LEN,8)[COP(Wrk_Main_Read_Buffer.DATA[4],Wrk_AdditionalLen,1) SWPB(Wrk_AdditionalLen,REVERSE,Wrk_AdditionalLen1) ADD(Wrk_AdditionalLen1,6,Wrk_AdditionaLenRead) ,GEQ(Wrk_AdditionaLenRead,8) GEQ(Wrk_Main_Read_Buffer.LEN,Wrk_AdditionaLenRead) [MID(Wrk_Main_Read_Buffer,Wrk_AdditionaLenRead,1,Wrk_ModbusPacket) ,DELETE(Wrk_Main_Read_Buffer,Wrk_AdditionaLenRead,1,Wrk_Main_Read_Buffer) ,OTE(Wrk_DataReceived) ] ];
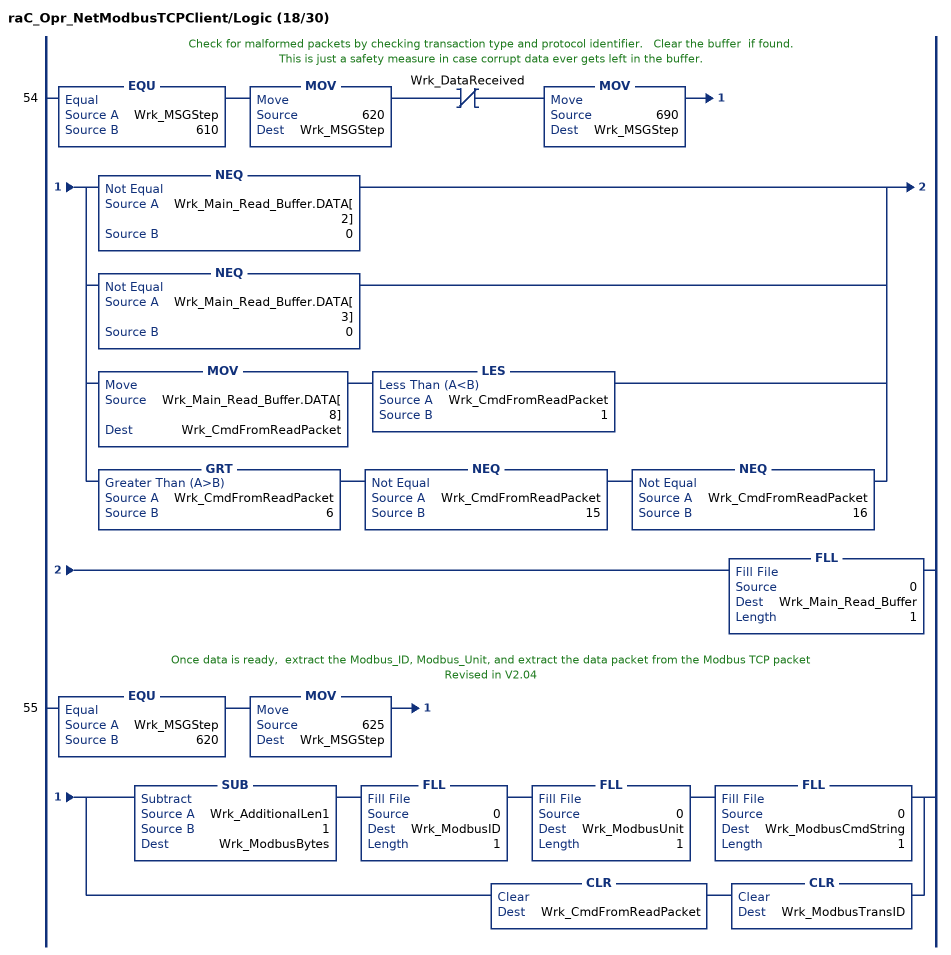
   // Check for malformed packets by checking transaction type and protocol identifier.   Clear the buffer  if found.
   // This is just a safety measure in case corrupt data ever gets left in the buffer.
   54: EQU(Wrk_MSGStep,610)MOV(620,Wrk_MSGStep)XIO(Wrk_DataReceived)MOV(690,Wrk_MSGStep)[NEQ(Wrk_Main_Read_Buffer.DATA[2],0) ,NEQ(Wrk_Main_Read_Buffer.DATA[3],0) ,MOV(Wrk_Main_Read_Buffer.DATA[8],Wrk_CmdFromReadPacket) LES(Wrk_CmdFromReadPacket,1) ,GRT(Wrk_CmdFromReadPacket,6) NEQ(Wrk_CmdFromReadPacket,15) NEQ(Wrk_CmdFromReadPacket,16) ]FLL(0,Wrk_Main_Read_Buffer,1);
   // Once data is ready,  extract the Modbus_ID, Modbus_Unit, and extract the data packet from the Modbus TCP packet
   // Revised in V2.04
   55: EQU(Wrk_MSGStep,620)MOV(625,Wrk_MSGStep)[SUB(Wrk_AdditionalLen1,1,Wrk_ModbusBytes) FLL(0,Wrk_ModbusID,1) FLL(0,Wrk_ModbusUnit,1) FLL(0,Wrk_ModbusCmdString,1) ,CLR(Wrk_CmdFromReadPacket) CLR(Wrk_ModbusTransID) ];
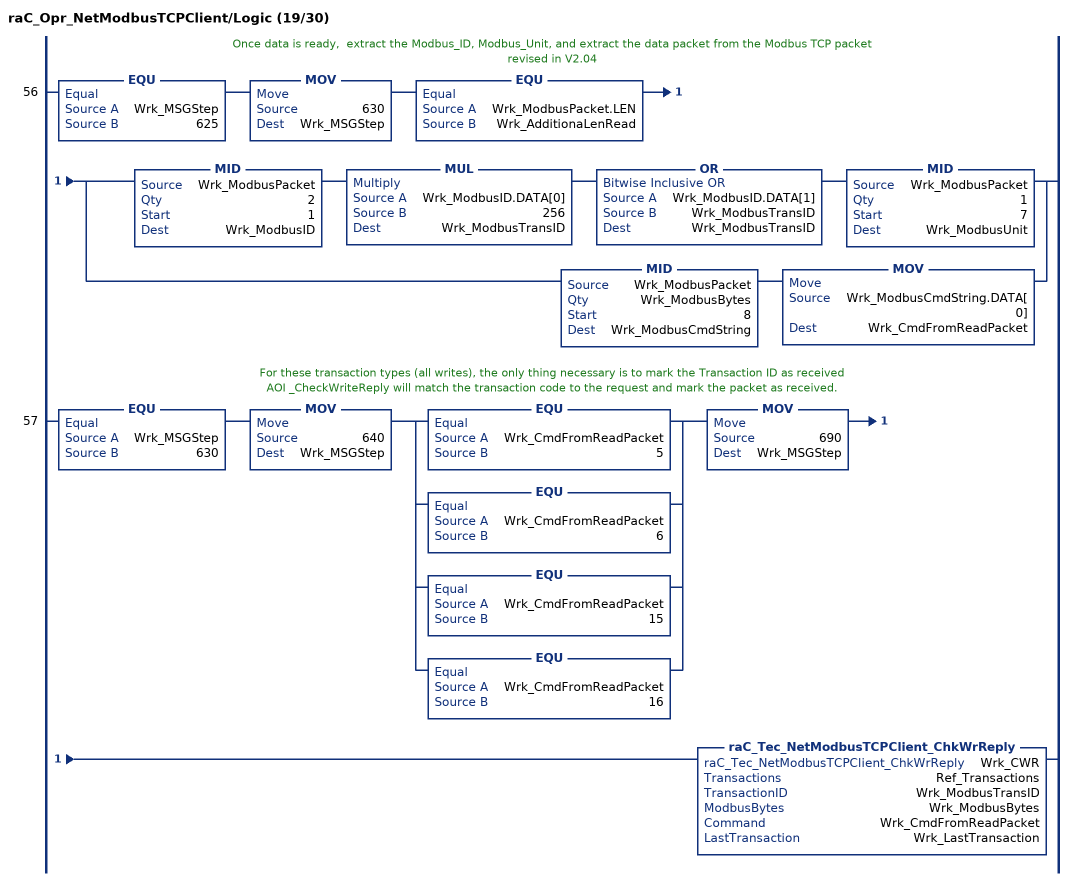
   // Once data is ready,  extract the Modbus_ID, Modbus_Unit, and extract the data packet from the Modbus TCP packet
   // revised in V2.04
   56: EQU(Wrk_MSGStep,625)MOV(630,Wrk_MSGStep)EQU(Wrk_ModbusPacket.LEN,Wrk_AdditionaLenRead)[MID(Wrk_ModbusPacket,2,1,Wrk_ModbusID) MUL(Wrk_ModbusID.DATA[0],256,Wrk_ModbusTransID) OR(Wrk_ModbusID.DATA[1],Wrk_ModbusTransID,Wrk_ModbusTransID) MID(Wrk_ModbusPacket,1,7,Wrk_ModbusUnit) ,MID(Wrk_ModbusPacket,Wrk_ModbusBytes,8,Wrk_ModbusCmdString) MOV(Wrk_ModbusCmdString.DATA[0],Wrk_CmdFromReadPacket) ];
   // For these transaction types (all writes), the only thing necessary is to mark the Transaction ID as received
   // AOI _CheckWriteReply will match the transaction code to the request and mark the packet as received.
   57: EQU(Wrk_MSGStep,630)MOV(640,Wrk_MSGStep)[EQU(Wrk_CmdFromReadPacket,5) ,EQU(Wrk_CmdFromReadPacket,6) ,EQU(Wrk_CmdFromReadPacket,15) ,EQU(Wrk_CmdFromReadPacket,16) ]MOV(690,Wrk_MSGStep)raC_Tec_NetModbusTCPClient_ChkWrReply(Wrk_CWR,Ref_Transactions,Wrk_ModbusTransID,Wrk_ModbusBytes,Wrk_CmdFromReadPacket,Wrk_LastTransaction);
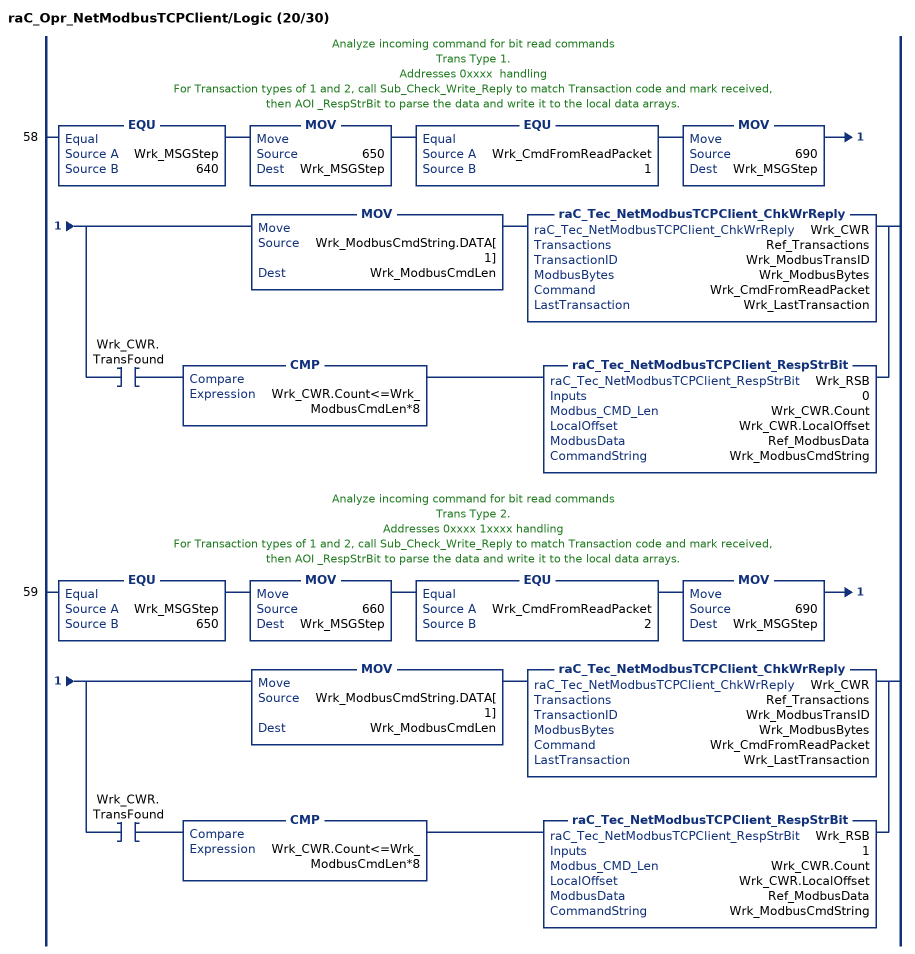
   // Analyze incoming command for bit read commands
   // Trans Type 1.
   // Addresses 0xxxx  handling
   // For Transaction types of 1 and 2, call Sub_Check_Write_Reply to match Transaction code and mark received,
   // then AOI _RespStrBit to parse the data and write it to the local data arrays.
   58: EQU(Wrk_MSGStep,640)MOV(650,Wrk_MSGStep)EQU(Wrk_CmdFromReadPacket,1)MOV(690,Wrk_MSGStep)[MOV(Wrk_ModbusCmdString.DATA[1],Wrk_ModbusCmdLen) raC_Tec_NetModbusTCPClient_ChkWrReply(Wrk_CWR,Ref_Transactions,Wrk_ModbusTransID,Wrk_ModbusBytes,Wrk_CmdFromReadPacket,Wrk_LastTransaction) ,XIC(Wrk_CWR.TransFound) CMP(Wrk_CWR.Count<=Wrk_ModbusCmdLen*8) raC_Tec_NetModbusTCPClient_RespStrBit(Wrk_RSB,0,Wrk_CWR.Count,Wrk_CWR.LocalOffset,Ref_ModbusData,Wrk_ModbusCmdString) ];
   // Analyze incoming command for bit read commands
   // Trans Type 2.
   // Addresses 0xxxx 1xxxx handling
   // For Transaction types of 1 and 2, call Sub_Check_Write_Reply to match Transaction code and mark received,
   // then AOI _RespStrBit to parse the data and write it to the local data arrays.
   59: EQU(Wrk_MSGStep,650)MOV(660,Wrk_MSGStep)EQU(Wrk_CmdFromReadPacket,2)MOV(690,Wrk_MSGStep)[MOV(Wrk_ModbusCmdString.DATA[1],Wrk_ModbusCmdLen) raC_Tec_NetModbusTCPClient_ChkWrReply(Wrk_CWR,Ref_Transactions,Wrk_ModbusTransID,Wrk_ModbusBytes,Wrk_CmdFromReadPacket,Wrk_LastTransaction) ,XIC(Wrk_CWR.TransFound) CMP(Wrk_CWR.Count<=Wrk_ModbusCmdLen*8) raC_Tec_NetModbusTCPClient_RespStrBit(Wrk_RSB,1,Wrk_CWR.Count,Wrk_CWR.LocalOffset,Ref_ModbusData,Wrk_ModbusCmdString) ];
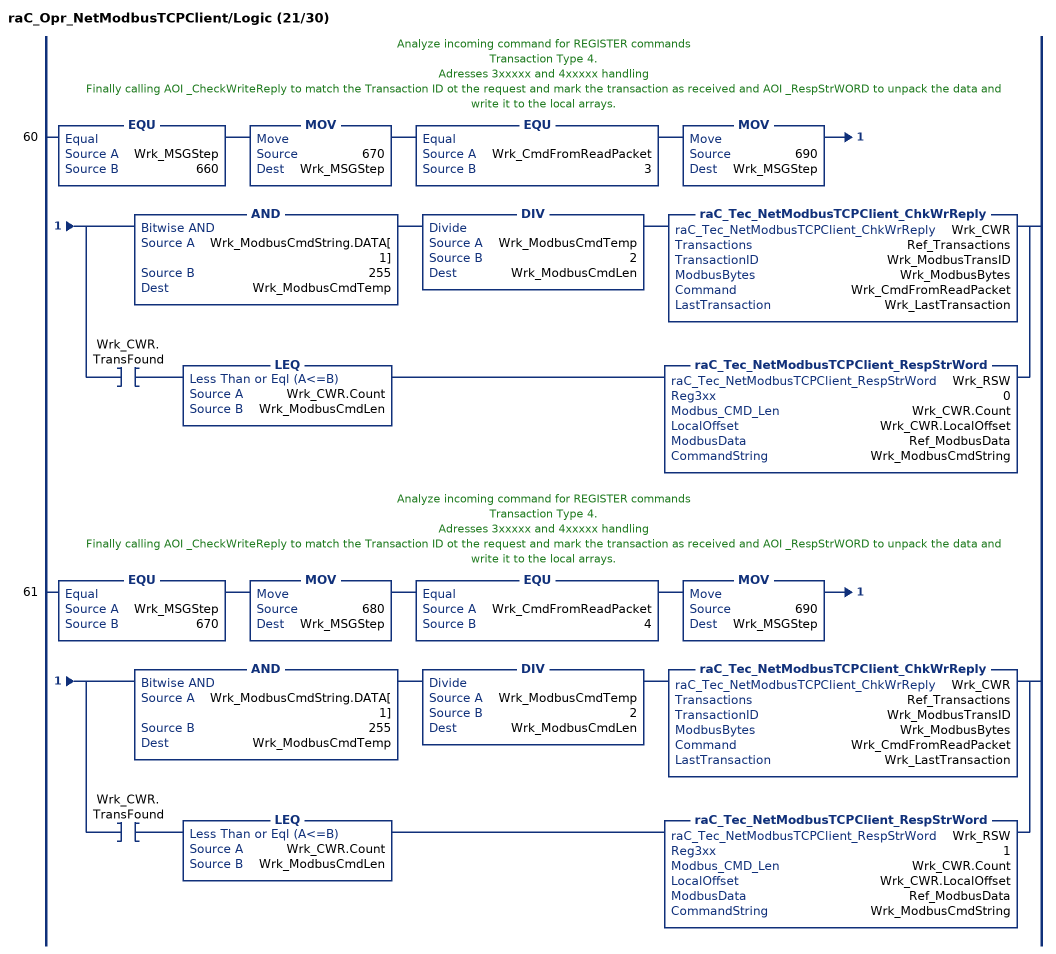
   // Analyze incoming command for REGISTER commands
   // Transaction Type 4.
   // Adresses 3xxxxx and 4xxxxx handling
   // Finally calling AOI _CheckWriteReply to match the Transaction ID ot the request and mark the transaction as received and AOI _RespStrWORD to unpack the data and write it to the local arrays.
   60: EQU(Wrk_MSGStep,660)MOV(670,Wrk_MSGStep)EQU(Wrk_CmdFromReadPacket,3)MOV(690,Wrk_MSGStep)[AND(Wrk_ModbusCmdString.DATA[1],255,Wrk_ModbusCmdTemp) DIV(Wrk_ModbusCmdTemp,2,Wrk_ModbusCmdLen) raC_Tec_NetModbusTCPClient_ChkWrReply(Wrk_CWR,Ref_Transactions,Wrk_ModbusTransID,Wrk_ModbusBytes,Wrk_CmdFromReadPacket,Wrk_LastTransaction) ,XIC(Wrk_CWR.TransFound) LEQ(Wrk_CWR.Count,Wrk_ModbusCmdLen) raC_Tec_NetModbusTCPClient_RespStrWord(Wrk_RSW,0,Wrk_CWR.Count,Wrk_CWR.LocalOffset,Ref_ModbusData,Wrk_ModbusCmdString) ];
   // Analyze incoming command for REGISTER commands
   // Transaction Type 4.
   // Adresses 3xxxxx and 4xxxxx handling
   // Finally calling AOI _CheckWriteReply to match the Transaction ID ot the request and mark the transaction as received and AOI _RespStrWORD to unpack the data and write it to the local arrays.
   61: EQU(Wrk_MSGStep,670)MOV(680,Wrk_MSGStep)EQU(Wrk_CmdFromReadPacket,4)MOV(690,Wrk_MSGStep)[AND(Wrk_ModbusCmdString.DATA[1],255,Wrk_ModbusCmdTemp) DIV(Wrk_ModbusCmdTemp,2,Wrk_ModbusCmdLen) raC_Tec_NetModbusTCPClient_ChkWrReply(Wrk_CWR,Ref_Transactions,Wrk_ModbusTransID,Wrk_ModbusBytes,Wrk_CmdFromReadPacket,Wrk_LastTransaction) ,XIC(Wrk_CWR.TransFound) LEQ(Wrk_CWR.Count,Wrk_ModbusCmdLen) raC_Tec_NetModbusTCPClient_RespStrWord(Wrk_RSW,1,Wrk_CWR.Count,Wrk_CWR.LocalOffset,Ref_ModbusData,Wrk_ModbusCmdString) ];
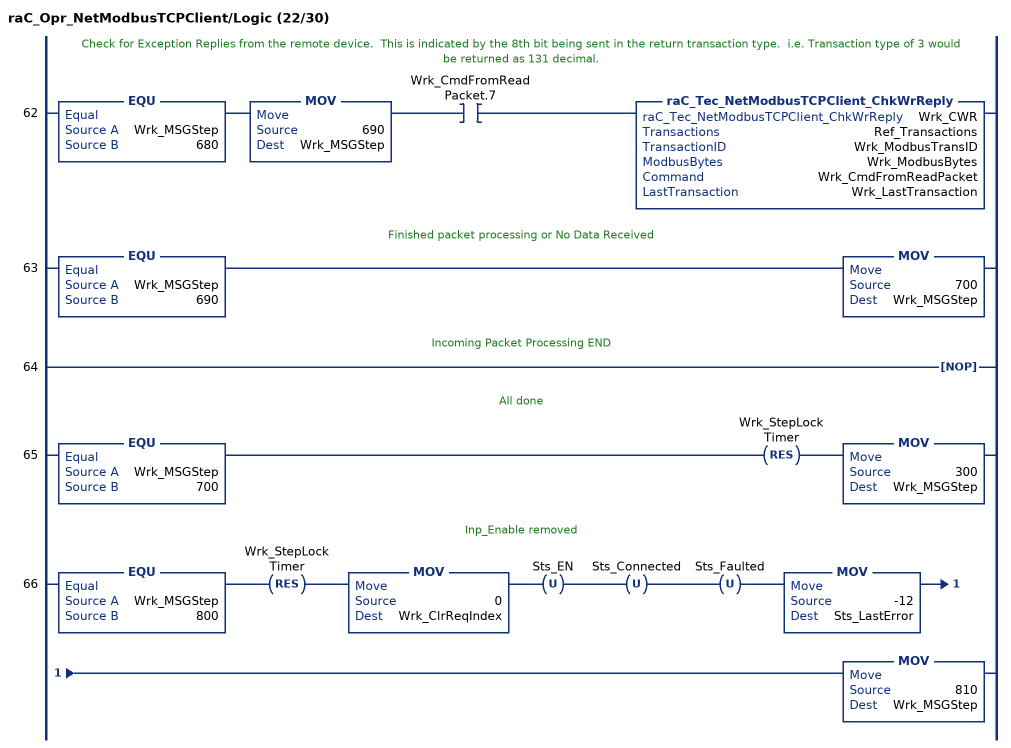
   // Check for Exception Replies from the remote device.  This is indicated by the 8th bit being sent in the return transaction type.  i.e. Transaction type of 3 would be returned as 131 decimal.
   62: EQU(Wrk_MSGStep,680)MOV(690,Wrk_MSGStep)XIC(Wrk_CmdFromReadPacket.7)raC_Tec_NetModbusTCPClient_ChkWrReply(Wrk_CWR,Ref_Transactions,Wrk_ModbusTransID,Wrk_ModbusBytes,Wrk_CmdFromReadPacket,Wrk_LastTransaction);
   // Finished packet processing or No Data Received
   63: EQU(Wrk_MSGStep,690)MOV(700,Wrk_MSGStep);
   // Incoming Packet Processing END
   64: NOP();
   // All done
   65: EQU(Wrk_MSGStep,700)RES(Wrk_StepLockTimer)MOV(300,Wrk_MSGStep);
   // Inp_Enable removed
   66: EQU(Wrk_MSGStep,800)RES(Wrk_StepLockTimer)MOV(0,Wrk_ClrReqIndex)OTU(Sts_EN)OTU(Sts_Connected)OTU(Sts_Faulted)MOV(-12,Sts_LastError)MOV(810,Wrk_MSGStep);
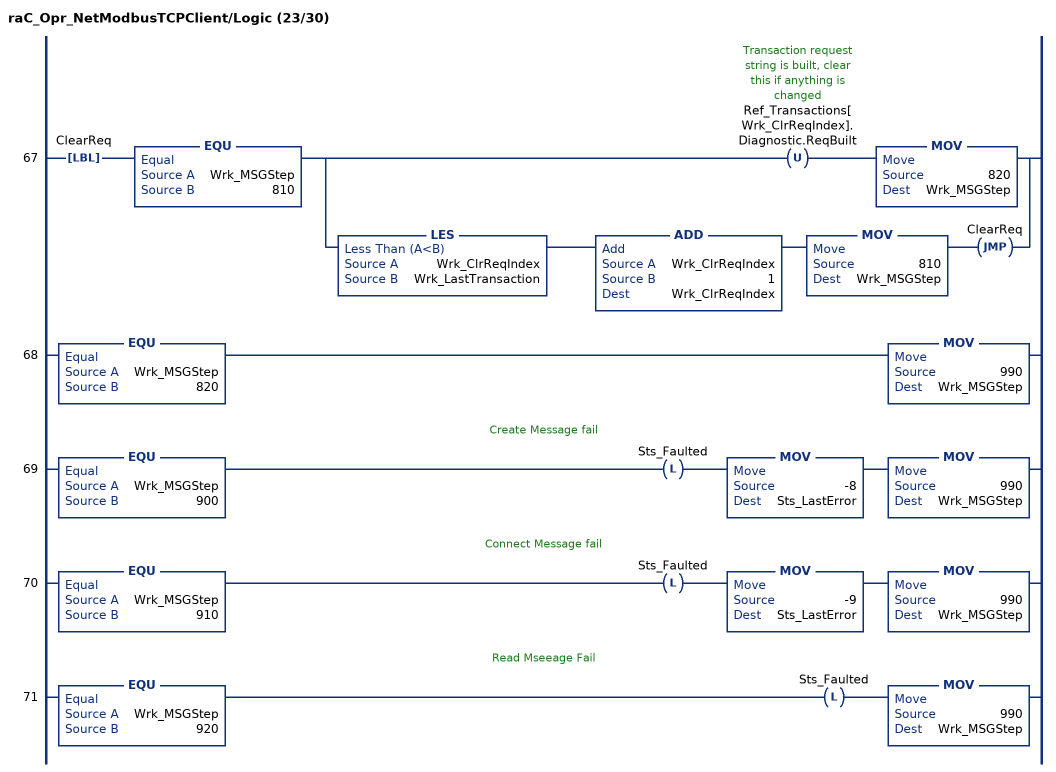
   67: LBL(ClearReq)EQU(Wrk_MSGStep,810)[OTU(Ref_Transactions[Wrk_ClrReqIndex].Diagnostic.ReqBuilt) MOV(820,Wrk_MSGStep) ,LES(Wrk_ClrReqIndex,Wrk_LastTransaction) ADD(Wrk_ClrReqIndex,1,Wrk_ClrReqIndex) MOV(810,Wrk_MSGStep) JMP(ClearReq) ];
   68: EQU(Wrk_MSGStep,820)MOV(990,Wrk_MSGStep);
   // Create Message fail
   69: EQU(Wrk_MSGStep,900)OTL(Sts_Faulted)MOV(-8,Sts_LastError)MOV(990,Wrk_MSGStep);
   // Connect Message fail
   70: EQU(Wrk_MSGStep,910)OTL(Sts_Faulted)MOV(-9,Sts_LastError)MOV(990,Wrk_MSGStep);
   // Read Mseeage Fail
   71: EQU(Wrk_MSGStep,920)OTL(Sts_Faulted)MOV(990,Wrk_MSGStep);
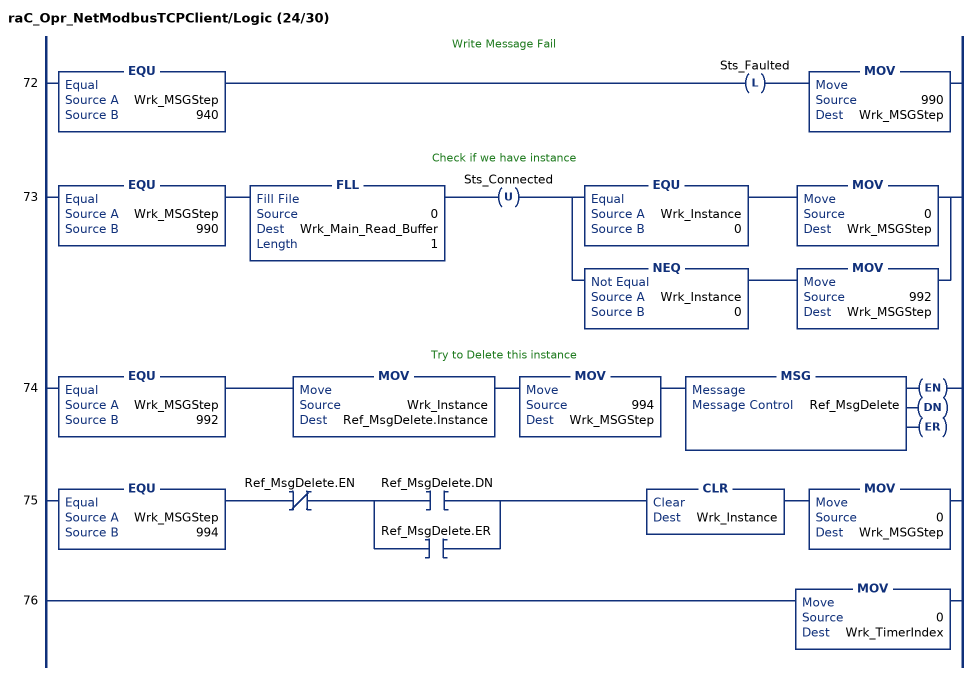
   // Write Message Fail
   72: EQU(Wrk_MSGStep,940)OTL(Sts_Faulted)MOV(990,Wrk_MSGStep);
   // Check if we have instance
   73: EQU(Wrk_MSGStep,990)FLL(0,Wrk_Main_Read_Buffer,1)OTU(Sts_Connected)[EQU(Wrk_Instance,0) MOV(0,Wrk_MSGStep) ,NEQ(Wrk_Instance,0) MOV(992,Wrk_MSGStep) ];
   // Try to Delete this instance
   74: EQU(Wrk_MSGStep,992)MOV(Wrk_Instance,Ref_MsgDelete.Instance)MOV(994,Wrk_MSGStep)MSG(Ref_MsgDelete);
   75: EQU(Wrk_MSGStep,994)XIO(Ref_MsgDelete.EN)[XIC(Ref_MsgDelete.DN) ,XIC(Ref_MsgDelete.ER) ]CLR(Wrk_Instance)MOV(0,Wrk_MSGStep);
   76: MOV(0,Wrk_TimerIndex);
